FUNCTION TryConvert_DATE_TO_ULINT : BOOL
VAR_INPUT
	in : DATE;
	out : REFERENCE TO ULINT;
END_VAR

out := DATE_TO_ULINT(in);
TryConvert_DATE_TO_ULINT := TRUE;

END_FUNCTION

(* stored: Version 1.1.0.1, ProductVersion 3.1.4024.12
   POU TryConvert_DATE_TO_ULINT: Id {6a1c6f0e-3d4a-428d-a010-88d9ed3fa644}, SpecialFunc None *)
